(* Logix 5000 project; controller DispersionPlc vendor 1 type 14 code 108 rev 34.11; software revision 34.01; part 12 of 22 *)
(* tags used below, declared in another part *)
   _Placeholder : DINT;
   dpt_4301_High : REAL;
   K200_PhaseTransfer : AStd_PLI;
   K200_PhaseTransfer_AOI : AStd_PLI_AOI;
   K200_PhaseTransfer_StepComplete : BOOL[32];
   K400_PhaseTransfer : AStd_PLI;
   LS_26_High : BOOL;
   LS_4301_High : BOOL;
   LS_4302_High : BOOL;
   MMI_T4301_Level : INT;
   PIDE_TCV_S47_1_AutoSP : REAL;
   SP : REAL;
   SPARE_I205 : ALIAS FOR Local:2:I.Data.5;
   SPARE_I410 : ALIAS FOR Local:4:I.Data.10;
   SPARE_I411 : ALIAS FOR Local:4:I.Data.11;
   SPARE_O607 : ALIAS FOR Local:6:O.Data.7;
   SPARE_O612 : ALIAS FOR Local:6:O.Data.12;
   TCV_S47_1_AutoCommand : REAL;
   TCV_S47_1_AutoSelected : BOOL;
   TIT_K200_3 : AStd_AnalogInput;
   TIT_K200_3_AOI : AStd_AI_AOI;
   TIT_K200_3_Val : REAL;
   TIT_K400_1 : AStd_AnalogInput;
   TIT_K400_1_AOI : AStd_AI_AOI;
   TIT_K400_1_Val : REAL;
   TIT_K400_3 : AStd_AnalogInput;
   TIT_K400_3_AOI : AStd_AI_AOI;
   TIT_S47_1_AOI : AStd_AI_AOI;
   TT_K200_2 : REAL;
   TT_K200_2_Raw : DINT;
   WIT_4302_1 : AStd_AnalogInput;
   XV_4301 : ALIAS FOR Local:5:O.Data.0;
   XV_4301_1 : AStd_VlvOC;
   XV_4301_1_AOI : AStd_VlvOC_AOI;
   XV_4301_1_IOpn : BOOL;
   XV_4301_1_OCls : BOOL;
   XV_4302 : ALIAS FOR Local:5:O.Data.1;
   XV_4302_1 : AStd_VlvOC;
   XV_4302_11 : AStd_VlvOC;
   XV_4302_11_AOI : AStd_VlvOC_AOI;
   XV_4302_11_IOpn : BOOL;
   XV_4302_11_OCls : BOOL;
   XV_4302_11Sol : BOOL;
   XV_4302_1_AOI : AStd_VlvOC_AOI;
   XV_4302_1_IOpn : BOOL;
   XV_4302_1_OCls : BOOL;
   XV_4302_7 : AStd_VlvOC;
   XV_4302_9 : AStd_VlvOC;
   XV_4302_9_AOI : AStd_VlvOC_AOI;
   XV_4302_9_IOpn : BOOL;
   XV_4302_9_OCls : BOOL;
   XV_K400_6 : AStd_VlvOC;
   XV_K400_6_AOI : AStd_VlvOC_AOI;
   XV_K400_6_IOpn : BOOL;
   XV_K400_6_OCls : BOOL;
   XV_K400_7 : AStd_VlvOC;
   XV_K400_7_AOI : AStd_VlvOC_AOI;
   XV_K400_7_IOpn : BOOL;
   XV_K400_7_OCls : BOOL;
   ZSC_4302 : ALIAS FOR Local:2:I.Data.3;
   ZSO_4301 : ALIAS FOR Local:2:I.Data.0;
(* PIDLoops, continued *)

ROUTINE PID_RO   (* function block diagram *)
   SHEET 1
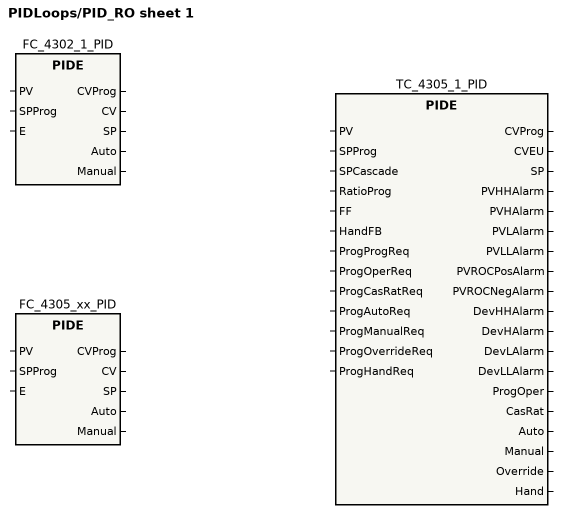
   FC_4302_1_PID : PIDE();   // unwired pins: PV SPProg CVProg CV SP E Auto Manual
   FC_4305_xx_PID : PIDE();   // unwired pins: PV SPProg CVProg CV SP E Auto Manual
   TC_4305_1_PID : PIDE();   // unwired pins: PV SPProg SPCascade RatioProg CVProg FF HandFB ProgProgReq ProgOperReq ProgCasRatReq ProgAutoReq ProgManualReq ProgOverrideReq ProgHandReq CVEU SP PVHHAlarm PVHAlarm PVLAlarm PVLLAlarm PVROCPosAlarm PVROCNegAlarm DevHHAlarm DevHAlarm DevLAlarm DevLLAlarm ProgOper CasRat Auto Manual Override Hand
END_ROUTINE

ROUTINE PID_TCV_S47_1   (* function block diagram *)
   SHEET 1
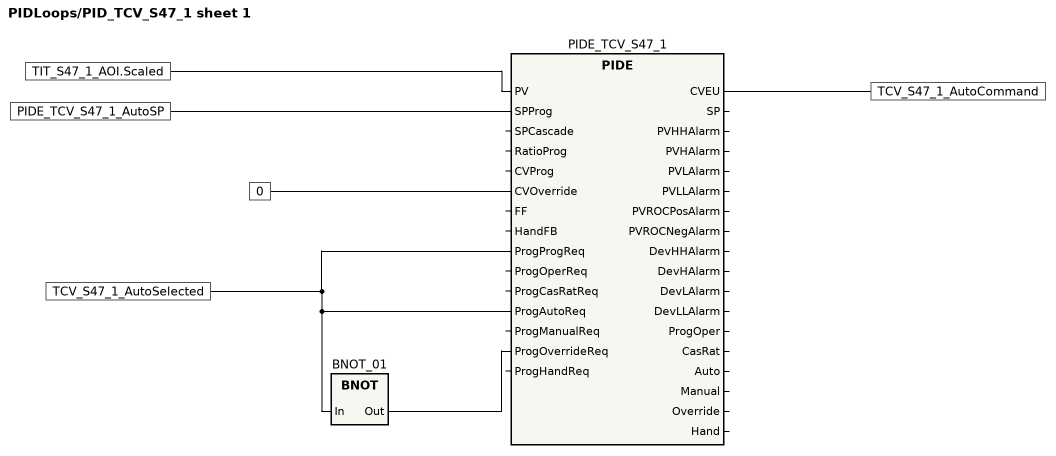
   BNOT_01 : BNOT(In := TCV_S47_1_AutoSelected);
   PIDE_TCV_S47_1 : PIDE(PV := TIT_S47_1_AOI.Scaled, SPProg := PIDE_TCV_S47_1_AutoSP, CVOverride := 0, ProgProgReq := TCV_S47_1_AutoSelected, ProgAutoReq := TCV_S47_1_AutoSelected, ProgOverrideReq := BNOT_01.Out);   // unwired pins: SPCascade RatioProg CVProg FF HandFB ProgOperReq ProgCasRatReq ProgManualReq ProgHandReq SP PVHHAlarm PVHAlarm PVLAlarm PVLLAlarm PVROCPosAlarm PVROCNegAlarm DevHHAlarm DevHAlarm DevLAlarm DevLLAlarm ProgOper CasRat Auto Manual Override Hand
   TCV_S47_1_AutoCommand := PIDE_TCV_S47_1.CVEU;
END_ROUTINE
END_PROGRAM

PROGRAM Simulation   (* main routine Main *)

ROUTINE Main   (* ladder *)
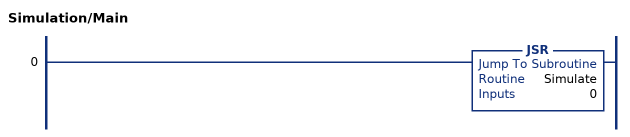
   0: JSR(Simulate,0);
END_ROUTINE

ROUTINE Simulate   (* ladder *)
END_ROUTINE
END_PROGRAM

PROGRAM Unit_K200   (* main routine MainRutine *)

ROUTINE Device_TIT_K200_3   (* ladder *)
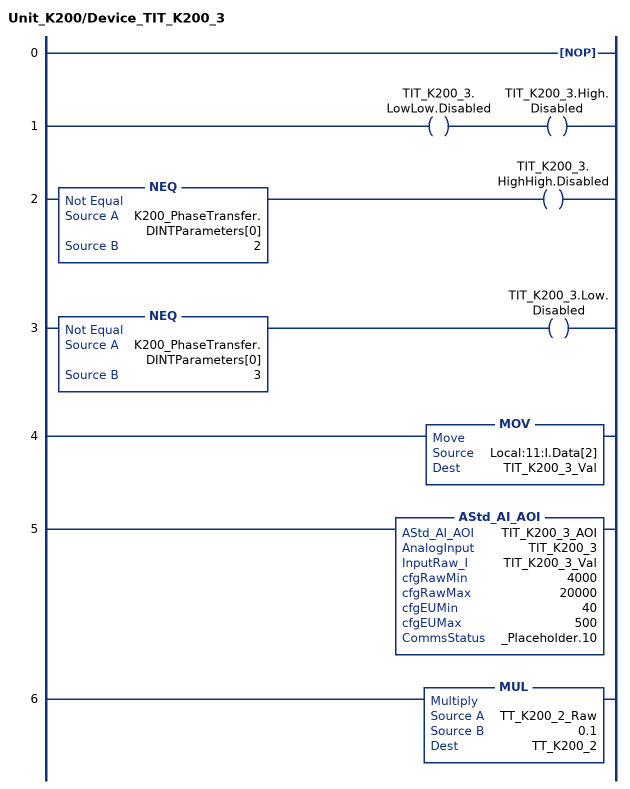
   0: NOP();
   1: OTE(TIT_K200_3.LowLow.Disabled)OTE(TIT_K200_3.High.Disabled);
   2: NEQ(K200_PhaseTransfer.DINTParameters[0],2)OTE(TIT_K200_3.HighHigh.Disabled);
   3: NEQ(K200_PhaseTransfer.DINTParameters[0],3)OTE(TIT_K200_3.Low.Disabled);
   4: MOV(Local:11:I.Data[2],TIT_K200_3_Val);
   5: AStd_AI_AOI(TIT_K200_3_AOI,TIT_K200_3,TIT_K200_3_Val,4000,20000,40,500,_Placeholder.10);
   6: MUL(TT_K200_2_Raw,0.1,TT_K200_2);
END_ROUTINE

ROUTINE Device_XV_4301_1   (* ladder *)
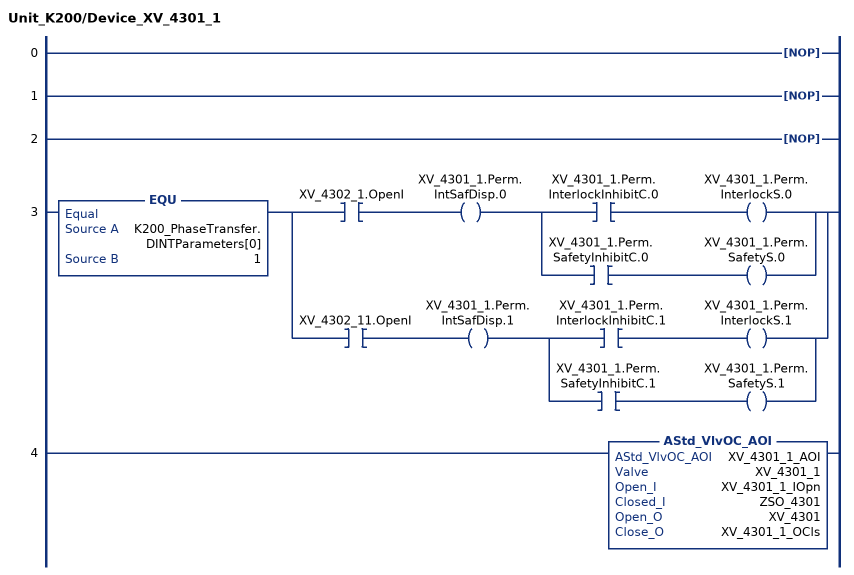
   0: NOP();
   1: NOP();
   2: NOP();
   3: EQU(K200_PhaseTransfer.DINTParameters[0],1)[XIC(XV_4302_1.OpenI) OTE(XV_4301_1.Perm.IntSafDisp.0) [XIC(XV_4301_1.Perm.InterlockInhibitC.0) OTE(XV_4301_1.Perm.InterlockS.0) ,XIC(XV_4301_1.Perm.SafetyInhibitC.0) OTE(XV_4301_1.Perm.SafetyS.0) ] ,XIC(XV_4302_11.OpenI) OTE(XV_4301_1.Perm.IntSafDisp.1) [XIC(XV_4301_1.Perm.InterlockInhibitC.1) OTE(XV_4301_1.Perm.InterlockS.1) ,XIC(XV_4301_1.Perm.SafetyInhibitC.1) OTE(XV_4301_1.Perm.SafetyS.1) ] ];
   4: AStd_VlvOC_AOI(XV_4301_1_AOI,XV_4301_1,XV_4301_1_IOpn,ZSO_4301,XV_4301,XV_4301_1_OCls);
END_ROUTINE

ROUTINE Device_XV_4302_1   (* ladder *)
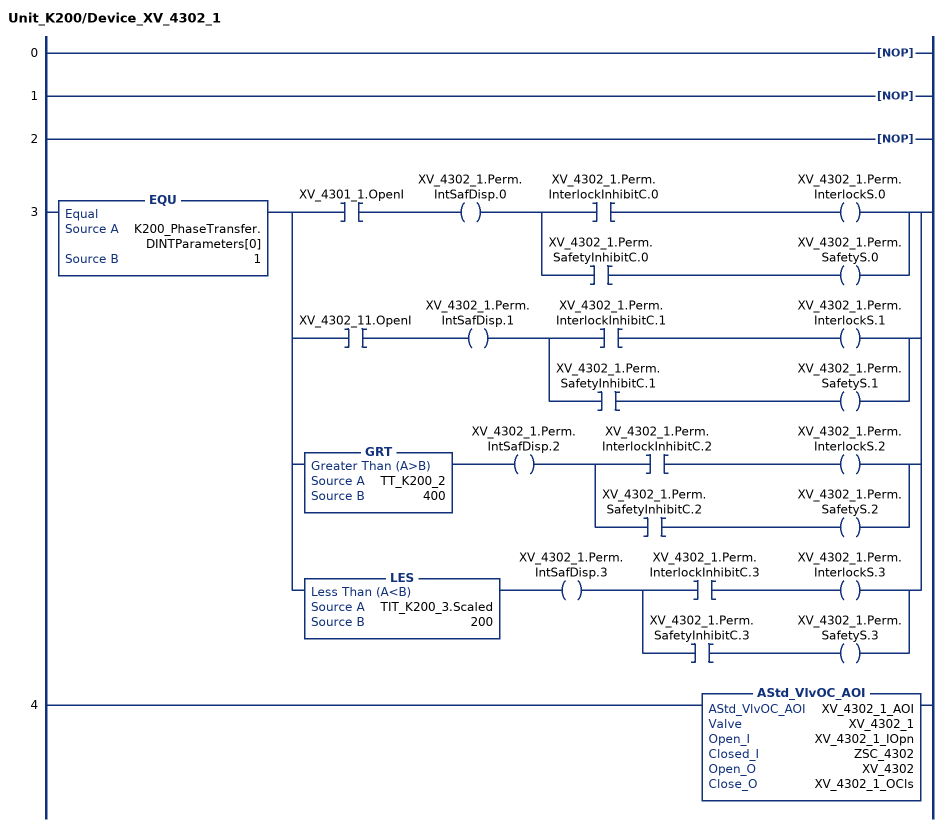
   0: NOP();
   1: NOP();
   2: NOP();
   3: EQU(K200_PhaseTransfer.DINTParameters[0],1)[XIC(XV_4301_1.OpenI) OTE(XV_4302_1.Perm.IntSafDisp.0) [XIC(XV_4302_1.Perm.InterlockInhibitC.0) OTE(XV_4302_1.Perm.InterlockS.0) ,XIC(XV_4302_1.Perm.SafetyInhibitC.0) OTE(XV_4302_1.Perm.SafetyS.0) ] ,XIC(XV_4302_11.OpenI) OTE(XV_4302_1.Perm.IntSafDisp.1) [XIC(XV_4302_1.Perm.InterlockInhibitC.1) OTE(XV_4302_1.Perm.InterlockS.1) ,XIC(XV_4302_1.Perm.SafetyInhibitC.1) OTE(XV_4302_1.Perm.SafetyS.1) ] ,GRT(TT_K200_2,400) OTE(XV_4302_1.Perm.IntSafDisp.2) [XIC(XV_4302_1.Perm.InterlockInhibitC.2) OTE(XV_4302_1.Perm.InterlockS.2) ,XIC(XV_4302_1.Perm.SafetyInhibitC.2) OTE(XV_4302_1.Perm.SafetyS.2) ] ,LES(TIT_K200_3.Scaled,200) OTE(XV_4302_1.Perm.IntSafDisp.3) [XIC(XV_4302_1.Perm.InterlockInhibitC.3) OTE(XV_4302_1.Perm.InterlockS.3) ,XIC(XV_4302_1.Perm.SafetyInhibitC.3) OTE(XV_4302_1.Perm.SafetyS.3) ] ];
   4: AStd_VlvOC_AOI(XV_4302_1_AOI,XV_4302_1,XV_4302_1_IOpn,ZSC_4302,XV_4302,XV_4302_1_OCls);
END_ROUTINE

ROUTINE Device_XV_4302_11   (* ladder *)
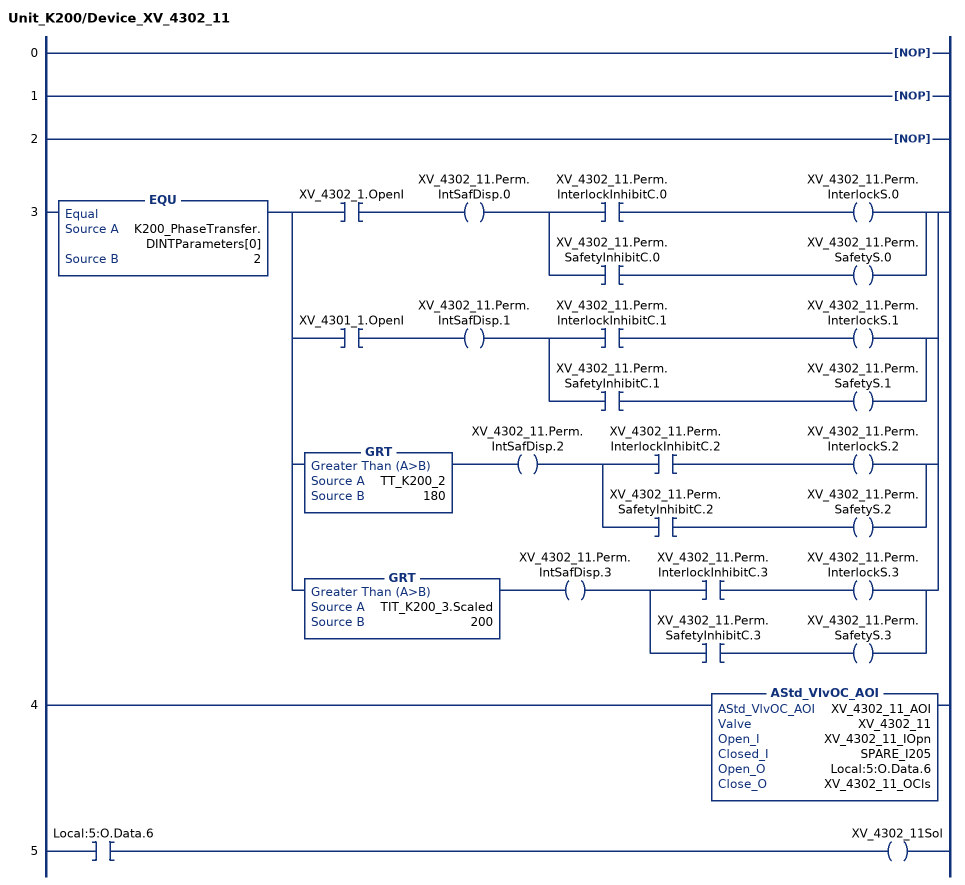
   0: NOP();
   1: NOP();
   2: NOP();
   3: EQU(K200_PhaseTransfer.DINTParameters[0],2)[XIC(XV_4302_1.OpenI) OTE(XV_4302_11.Perm.IntSafDisp.0) [XIC(XV_4302_11.Perm.InterlockInhibitC.0) OTE(XV_4302_11.Perm.InterlockS.0) ,XIC(XV_4302_11.Perm.SafetyInhibitC.0) OTE(XV_4302_11.Perm.SafetyS.0) ] ,XIC(XV_4301_1.OpenI) OTE(XV_4302_11.Perm.IntSafDisp.1) [XIC(XV_4302_11.Perm.InterlockInhibitC.1) OTE(XV_4302_11.Perm.InterlockS.1) ,XIC(XV_4302_11.Perm.SafetyInhibitC.1) OTE(XV_4302_11.Perm.SafetyS.1) ] ,GRT(TT_K200_2,180) OTE(XV_4302_11.Perm.IntSafDisp.2) [XIC(XV_4302_11.Perm.InterlockInhibitC.2) OTE(XV_4302_11.Perm.InterlockS.2) ,XIC(XV_4302_11.Perm.SafetyInhibitC.2) OTE(XV_4302_11.Perm.SafetyS.2) ] ,GRT(TIT_K200_3.Scaled,200) OTE(XV_4302_11.Perm.IntSafDisp.3) [XIC(XV_4302_11.Perm.InterlockInhibitC.3) OTE(XV_4302_11.Perm.InterlockS.3) ,XIC(XV_4302_11.Perm.SafetyInhibitC.3) OTE(XV_4302_11.Perm.SafetyS.3) ] ];
   4: AStd_VlvOC_AOI(XV_4302_11_AOI,XV_4302_11,XV_4302_11_IOpn,SPARE_I205,Local:5:O.Data.6,XV_4302_11_OCls);
   5: XIC(Local:5:O.Data.6)OTE(XV_4302_11Sol);
END_ROUTINE

ROUTINE MainRutine   (* ladder *)
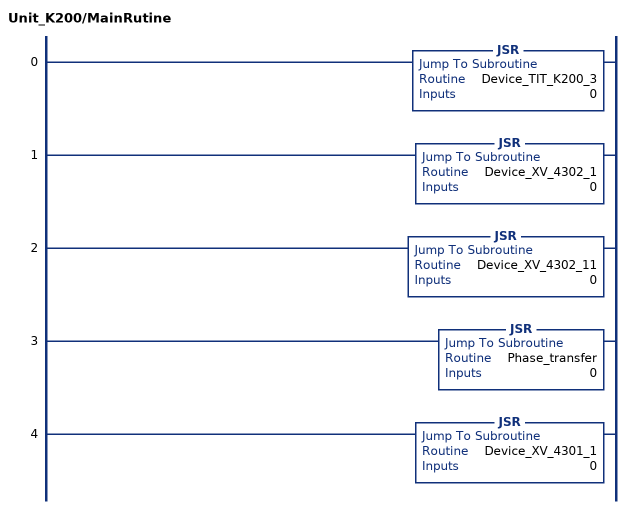
   0: JSR(Device_TIT_K200_3,0);
   1: JSR(Device_XV_4302_1,0);
   2: JSR(Device_XV_4302_11,0);
   3: JSR(Phase_transfer,0);
   4: JSR(Device_XV_4301_1,0);
END_ROUTINE

ROUTINE Phase_transfer   (* ladder *)
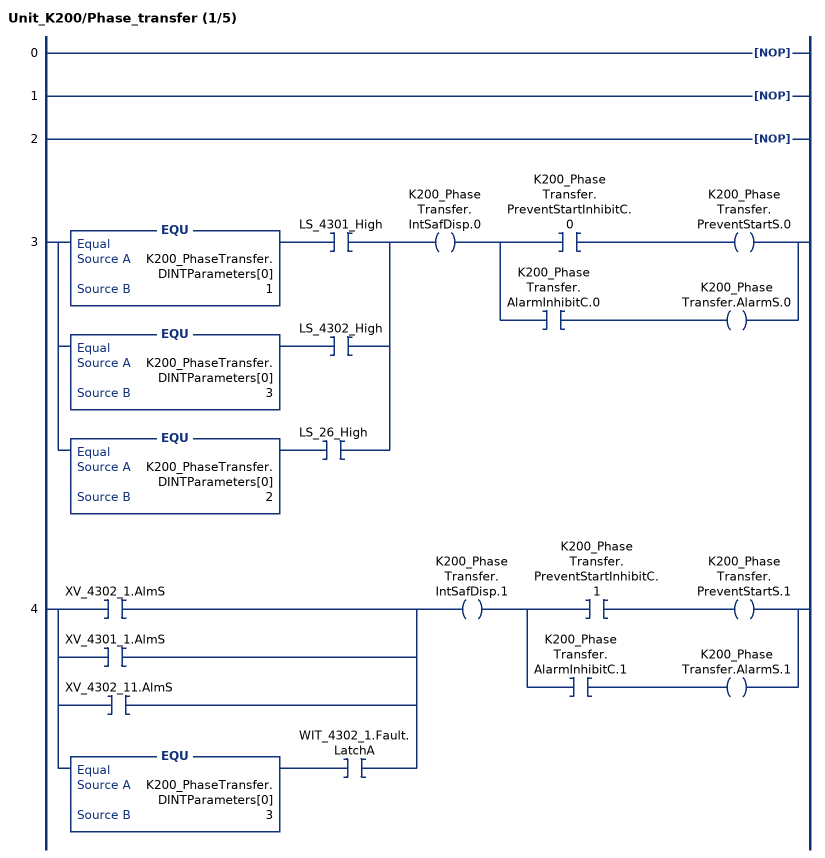
   0: NOP();
   1: NOP();
   2: NOP();
   3: [EQU(K200_PhaseTransfer.DINTParameters[0],1) XIC(LS_4301_High) ,EQU(K200_PhaseTransfer.DINTParameters[0],3) XIC(LS_4302_High) ,EQU(K200_PhaseTransfer.DINTParameters[0],2) XIC(LS_26_High) ]OTE(K200_PhaseTransfer.IntSafDisp.0)[XIC(K200_PhaseTransfer.PreventStartInhibitC.0) OTE(K200_PhaseTransfer.PreventStartS.0) ,XIC(K200_PhaseTransfer.AlarmInhibitC.0) OTE(K200_PhaseTransfer.AlarmS.0) ];
   4: [XIC(XV_4302_1.AlmS) ,XIC(XV_4301_1.AlmS) ,XIC(XV_4302_11.AlmS) ,EQU(K200_PhaseTransfer.DINTParameters[0],3) XIC(WIT_4302_1.Fault.LatchA) ]OTE(K200_PhaseTransfer.IntSafDisp.1)[XIC(K200_PhaseTransfer.PreventStartInhibitC.1) OTE(K200_PhaseTransfer.PreventStartS.1) ,XIC(K200_PhaseTransfer.AlarmInhibitC.1) OTE(K200_PhaseTransfer.AlarmS.1) ];
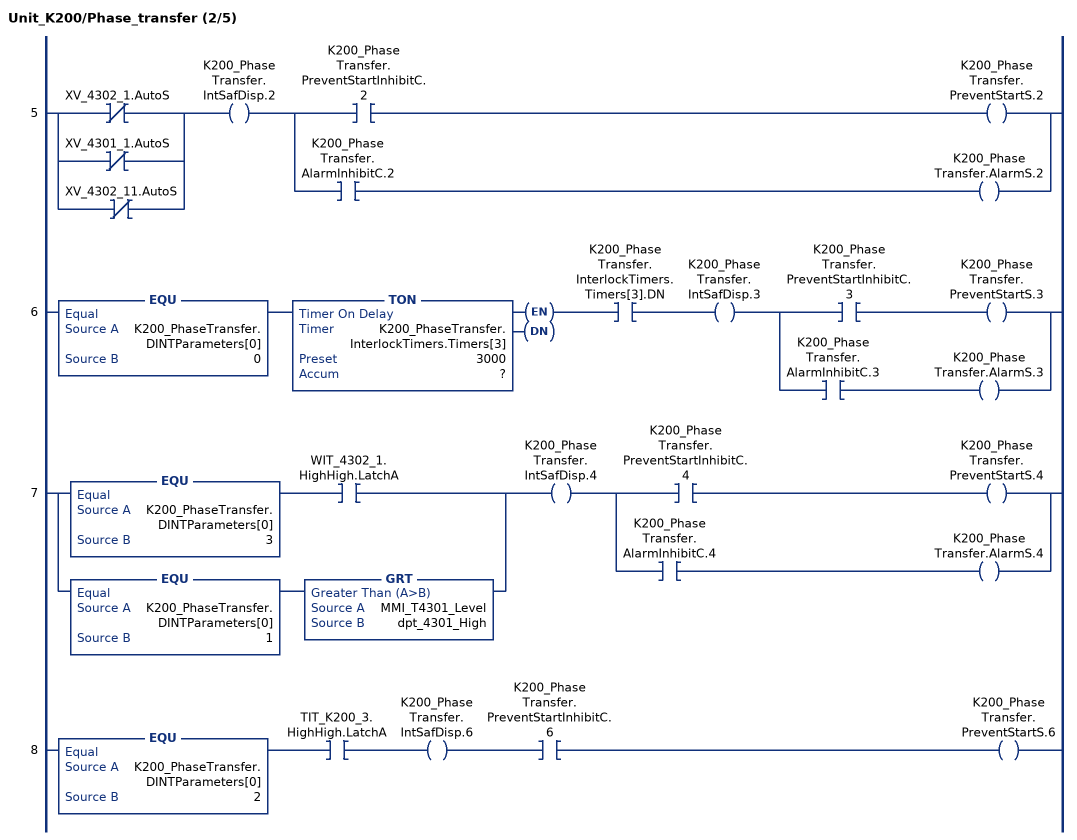
   5: [XIO(XV_4302_1.AutoS) ,XIO(XV_4301_1.AutoS) ,XIO(XV_4302_11.AutoS) ]OTE(K200_PhaseTransfer.IntSafDisp.2)[XIC(K200_PhaseTransfer.PreventStartInhibitC.2) OTE(K200_PhaseTransfer.PreventStartS.2) ,XIC(K200_PhaseTransfer.AlarmInhibitC.2) OTE(K200_PhaseTransfer.AlarmS.2) ];
   6: EQU(K200_PhaseTransfer.DINTParameters[0],0)TON(K200_PhaseTransfer.InterlockTimers.Timers[3],?,?)XIC(K200_PhaseTransfer.InterlockTimers.Timers[3].DN)OTE(K200_PhaseTransfer.IntSafDisp.3)[XIC(K200_PhaseTransfer.PreventStartInhibitC.3) OTE(K200_PhaseTransfer.PreventStartS.3) ,XIC(K200_PhaseTransfer.AlarmInhibitC.3) OTE(K200_PhaseTransfer.AlarmS.3) ];
   7: [EQU(K200_PhaseTransfer.DINTParameters[0],3) XIC(WIT_4302_1.HighHigh.LatchA) ,EQU(K200_PhaseTransfer.DINTParameters[0],1) GRT(MMI_T4301_Level,dpt_4301_High) ]OTE(K200_PhaseTransfer.IntSafDisp.4)[XIC(K200_PhaseTransfer.PreventStartInhibitC.4) OTE(K200_PhaseTransfer.PreventStartS.4) ,XIC(K200_PhaseTransfer.AlarmInhibitC.4) OTE(K200_PhaseTransfer.AlarmS.4) ];
   8: EQU(K200_PhaseTransfer.DINTParameters[0],2)XIC(TIT_K200_3.HighHigh.LatchA)OTE(K200_PhaseTransfer.IntSafDisp.6)XIC(K200_PhaseTransfer.PreventStartInhibitC.6)OTE(K200_PhaseTransfer.PreventStartS.6);
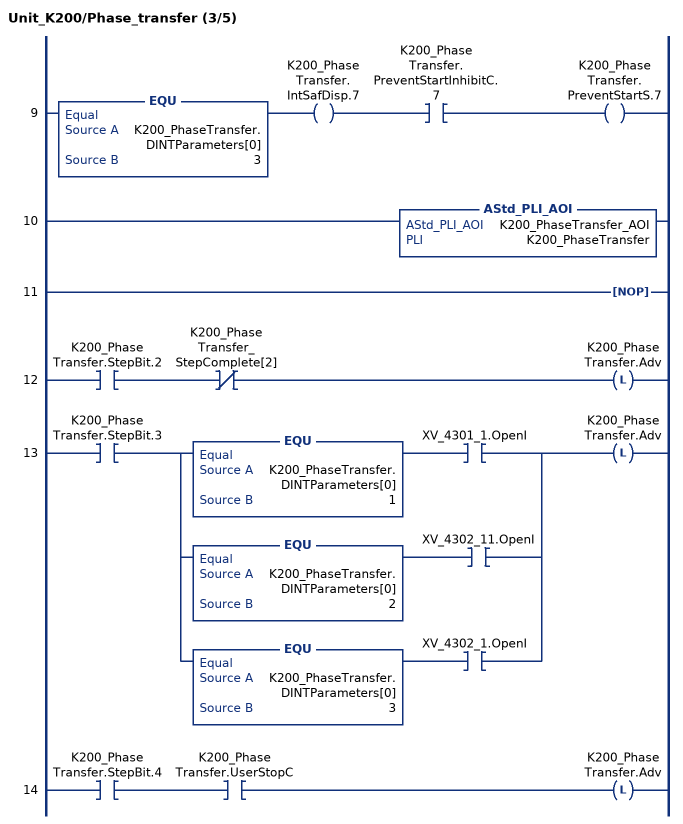
   9: EQU(K200_PhaseTransfer.DINTParameters[0],3)OTE(K200_PhaseTransfer.IntSafDisp.7)XIC(K200_PhaseTransfer.PreventStartInhibitC.7)OTE(K200_PhaseTransfer.PreventStartS.7);
   10: AStd_PLI_AOI(K200_PhaseTransfer_AOI,K200_PhaseTransfer);
   11: NOP();
   12: XIC(K200_PhaseTransfer.StepBit.2)XIO(K200_PhaseTransfer_StepComplete[2])OTL(K200_PhaseTransfer.Adv);
   13: XIC(K200_PhaseTransfer.StepBit.3)[EQU(K200_PhaseTransfer.DINTParameters[0],1) XIC(XV_4301_1.OpenI) ,EQU(K200_PhaseTransfer.DINTParameters[0],2) XIC(XV_4302_11.OpenI) ,EQU(K200_PhaseTransfer.DINTParameters[0],3) XIC(XV_4302_1.OpenI) ]OTL(K200_PhaseTransfer.Adv);
   14: XIC(K200_PhaseTransfer.StepBit.4)XIC(K200_PhaseTransfer.UserStopC)OTL(K200_PhaseTransfer.Adv);
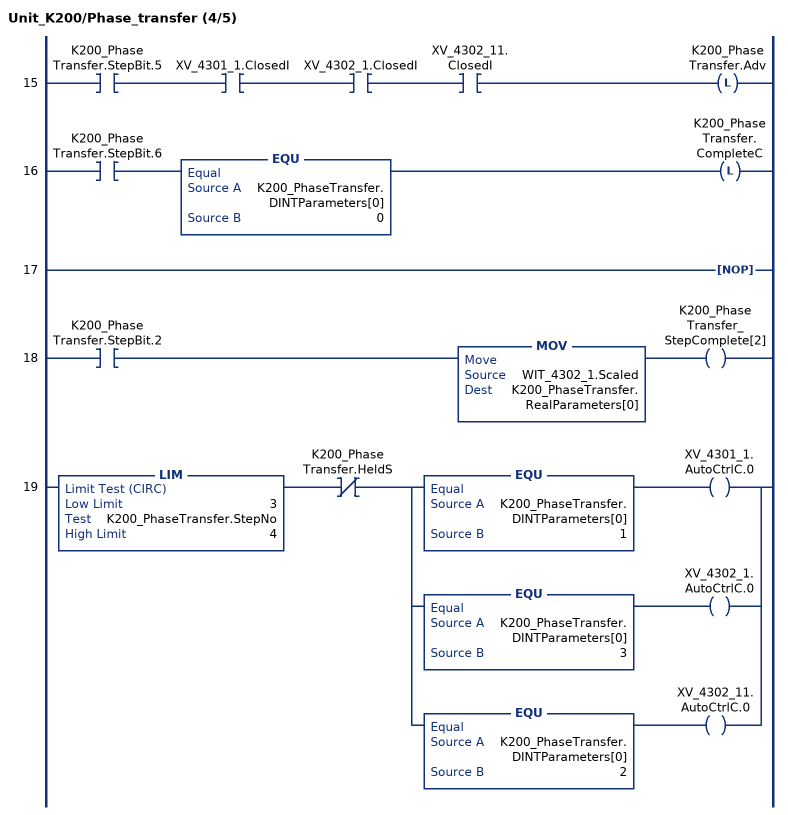
   15: XIC(K200_PhaseTransfer.StepBit.5)XIC(XV_4301_1.ClosedI)XIC(XV_4302_1.ClosedI)XIC(XV_4302_11.ClosedI)OTL(K200_PhaseTransfer.Adv);
   16: XIC(K200_PhaseTransfer.StepBit.6)EQU(K200_PhaseTransfer.DINTParameters[0],0)OTL(K200_PhaseTransfer.CompleteC);
   17: NOP();
   18: XIC(K200_PhaseTransfer.StepBit.2)MOV(WIT_4302_1.Scaled,K200_PhaseTransfer.RealParameters[0])OTE(K200_PhaseTransfer_StepComplete[2]);
   19: LIM(3,K200_PhaseTransfer.StepNo,4)XIO(K200_PhaseTransfer.HeldS)[EQU(K200_PhaseTransfer.DINTParameters[0],1) OTE(XV_4301_1.AutoCtrlC.0) ,EQU(K200_PhaseTransfer.DINTParameters[0],3) OTE(XV_4302_1.AutoCtrlC.0) ,EQU(K200_PhaseTransfer.DINTParameters[0],2) OTE(XV_4302_11.AutoCtrlC.0) ];
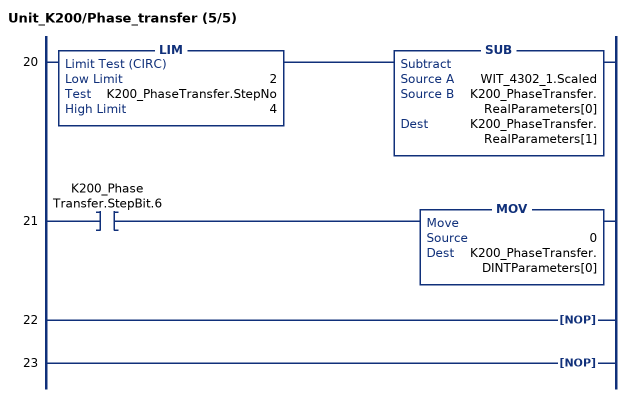
   20: LIM(2,K200_PhaseTransfer.StepNo,4)SUB(WIT_4302_1.Scaled,K200_PhaseTransfer.RealParameters[0],K200_PhaseTransfer.RealParameters[1]);
   21: XIC(K200_PhaseTransfer.StepBit.6)MOV(0,K200_PhaseTransfer.DINTParameters[0]);
   22: NOP();
   23: NOP();
END_ROUTINE
END_PROGRAM

PROGRAM Unit_K400   (* main routine MainRoutine *)

ROUTINE Devic_TIT_K400_3   (* ladder *)
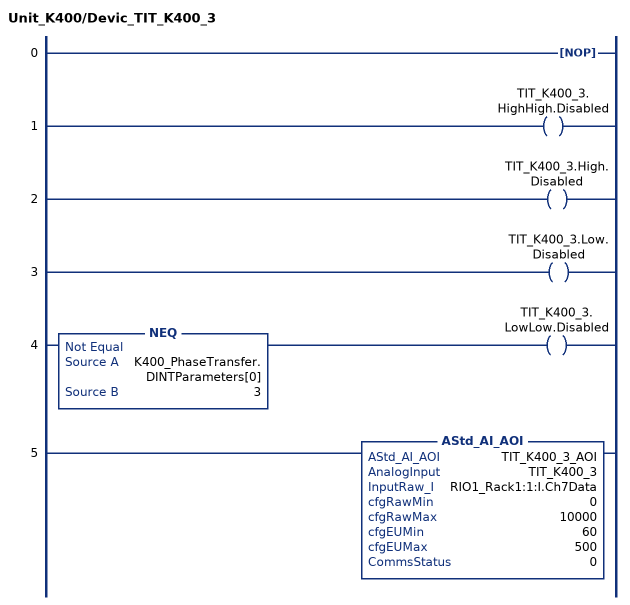
   0: NOP();
   1: OTE(TIT_K400_3.HighHigh.Disabled);
   2: OTE(TIT_K400_3.High.Disabled);
   3: OTE(TIT_K400_3.Low.Disabled);
   4: NEQ(K400_PhaseTransfer.DINTParameters[0],3)OTE(TIT_K400_3.LowLow.Disabled);
   5: AStd_AI_AOI(TIT_K400_3_AOI,TIT_K400_3,RIO1_Rack1:1:I.Ch7Data,0,10000,60,500,0);
END_ROUTINE

ROUTINE Device_TIT_K400_1   (* ladder *)
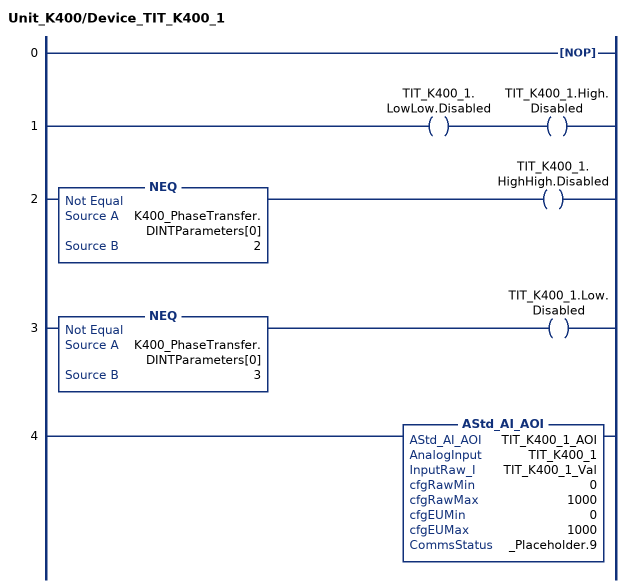
   0: NOP();
   1: OTE(TIT_K400_1.LowLow.Disabled)OTE(TIT_K400_1.High.Disabled);
   2: NEQ(K400_PhaseTransfer.DINTParameters[0],2)OTE(TIT_K400_1.HighHigh.Disabled);
   3: NEQ(K400_PhaseTransfer.DINTParameters[0],3)OTE(TIT_K400_1.Low.Disabled);
   4: AStd_AI_AOI(TIT_K400_1_AOI,TIT_K400_1,TIT_K400_1_Val,0,1000,0,1000,_Placeholder.9);
END_ROUTINE

ROUTINE Device_XV_4302_9   (* ladder *)
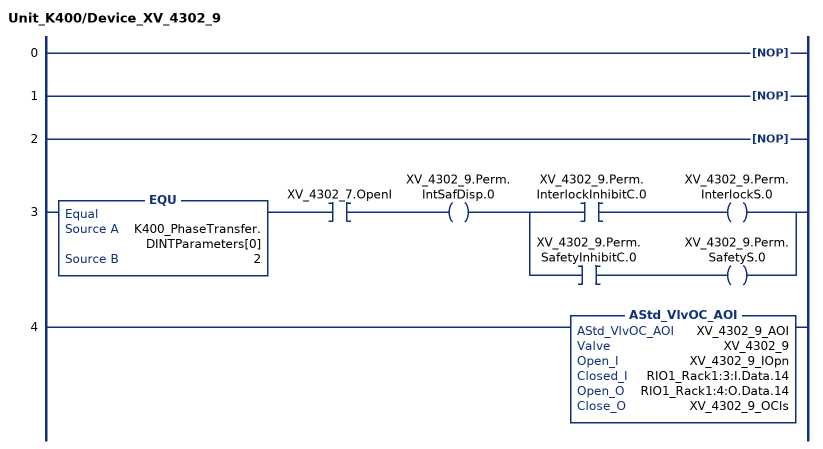
   0: NOP();
   1: NOP();
   2: NOP();
   3: EQU(K400_PhaseTransfer.DINTParameters[0],2)XIC(XV_4302_7.OpenI)OTE(XV_4302_9.Perm.IntSafDisp.0)[XIC(XV_4302_9.Perm.InterlockInhibitC.0) OTE(XV_4302_9.Perm.InterlockS.0) ,XIC(XV_4302_9.Perm.SafetyInhibitC.0) OTE(XV_4302_9.Perm.SafetyS.0) ];
   4: AStd_VlvOC_AOI(XV_4302_9_AOI,XV_4302_9,XV_4302_9_IOpn,RIO1_Rack1:3:I.Data.14,RIO1_Rack1:4:O.Data.14,XV_4302_9_OCls);
END_ROUTINE

ROUTINE Device_XV_K400_6   (* ladder *)
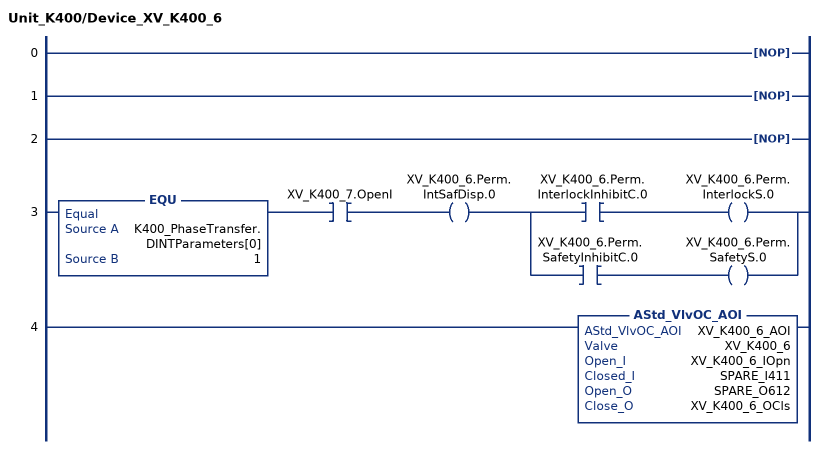
   0: NOP();
   1: NOP();
   2: NOP();
   3: EQU(K400_PhaseTransfer.DINTParameters[0],1)XIC(XV_K400_7.OpenI)OTE(XV_K400_6.Perm.IntSafDisp.0)[XIC(XV_K400_6.Perm.InterlockInhibitC.0) OTE(XV_K400_6.Perm.InterlockS.0) ,XIC(XV_K400_6.Perm.SafetyInhibitC.0) OTE(XV_K400_6.Perm.SafetyS.0) ];
   4: AStd_VlvOC_AOI(XV_K400_6_AOI,XV_K400_6,XV_K400_6_IOpn,SPARE_I411,SPARE_O612,XV_K400_6_OCls);
END_ROUTINE

ROUTINE Device_XV_K400_7   (* ladder *)
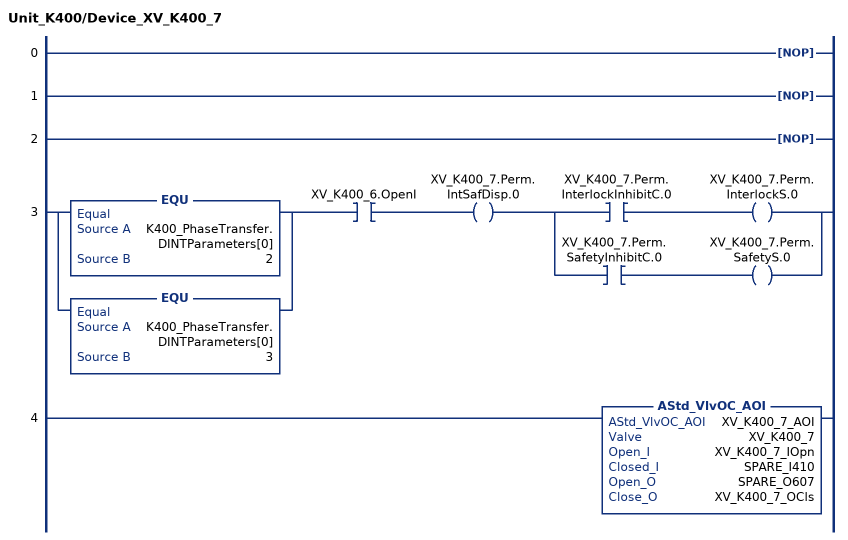
   0: NOP();
   1: NOP();
   2: NOP();
   3: [EQU(K400_PhaseTransfer.DINTParameters[0],2) ,EQU(K400_PhaseTransfer.DINTParameters[0],3) ]XIC(XV_K400_6.OpenI)OTE(XV_K400_7.Perm.IntSafDisp.0)[XIC(XV_K400_7.Perm.InterlockInhibitC.0) OTE(XV_K400_7.Perm.InterlockS.0) ,XIC(XV_K400_7.Perm.SafetyInhibitC.0) OTE(XV_K400_7.Perm.SafetyS.0) ];
   4: AStd_VlvOC_AOI(XV_K400_7_AOI,XV_K400_7,XV_K400_7_IOpn,SPARE_I410,SPARE_O607,XV_K400_7_OCls);
END_ROUTINE
